// TIA Portal project "empty" (V15.1)

(* hardware
DEVICE "S7-1200 station_1"  S7-1200 Station
   slot 0: "Rack_0"  S7-1200 Rack  Rack  V1.0
   slot 1: "PLC_1"  CPU 1217C DC/DC/DC  6ES7 217-1AG40-0XB0  V4.1
*)

// ===== PLC "PLC_1"  CPU 1217C DC/DC/DC =====

VAR_GLOBAL   // PLC tag table "Default tag table"
   "b1_Pulse" AT %Q0.1 : Bool;
   "b1_Direction" AT %Q0.5 : Bool;
   "Tag_1" AT %M0.0 : Bool;
   "Tag_2" AT %M0.1 : Bool;
   "System_Byte" AT %MB0 : Byte;
   "FirstScan" AT %M0.0 : Bool;
   "DiagStatusUpdate" AT %M0.1 : Bool;
   "AlwaysTRUE" AT %M0.2 : Bool;
   "AlwaysFALSE" AT %M0.3 : Bool;
   "Clock_Byte" AT %MB1 : Byte;
   "Clock_10Hz" AT %M1.0 : Bool;
   "Clock_5Hz" AT %M1.1 : Bool;
   "Clock_2.5Hz" AT %M1.2 : Bool;
   "Clock_2Hz" AT %M1.3 : Bool;
   "Clock_1.25Hz" AT %M1.4 : Bool;
   "Clock_1Hz" AT %M1.5 : Bool;
   "Clock_0.625Hz" AT %M1.6 : Bool;
   "Clock_0.5Hz" AT %M1.7 : Bool;
END_VAR

DATA_BLOCK "b1"   // DB1, Motion_DB
{ S7_Optimized_Access := 'TRUE' }
AUTHOR : SIMATIC
FAMILY : BasicMC
NAME : TO_PosAx
VERSION : 5.0
// stored: InstanceOfName TO_PositioningAxis
"TO_PositioningAxis"
BEGIN
   // Axis.LengthUnitNormalized.Distance = 1005
   // Axis.DirectionOutputEnabledCU = TRUE
   // Axis.OnlinePtoModeCU = 16#0000_0002
   // Axis.SelectedChannel2EnumCU = %Q0.5
   // Axis.SelectedChannel1EnumCU = %Q0.1
   // Pulse.MinDeltaDeltaFrequencyCU = 0.004
   // Pulse.MaxDeltaDeltaFrequencyCU = 1.0E+10
   // Pulse.MinDeltaFrequencyCU = 0.005
   // Pulse.MaxDeltaFrequencyCU = 9.5E+9
   // Pulse.MinFrequencyCU = 1.0
   // Pulse.MaxFrequencyCU = 1.0E+6
   // Pulse.OutputSourceCU = 16#0000_0000
   // Axis.SelectPTO = 0
   // Axis.LengthUnit.LastDistance = 1005
END_DATA_BLOCK

ORGANIZATION_BLOCK "Main"   // OB1, LAD, ProgramCycle
TITLE = "Main Program Sweep (Cycle)"
{ S7_Optimized_Access := 'TRUE' }
VERSION : 0.1
   VAR_INPUT
      Initial_Call : Bool;   // Initial call of this OB
      Remanence : Bool;   // =True, if remanent data are available
   END_VAR
BEGIN

REGION Network 1
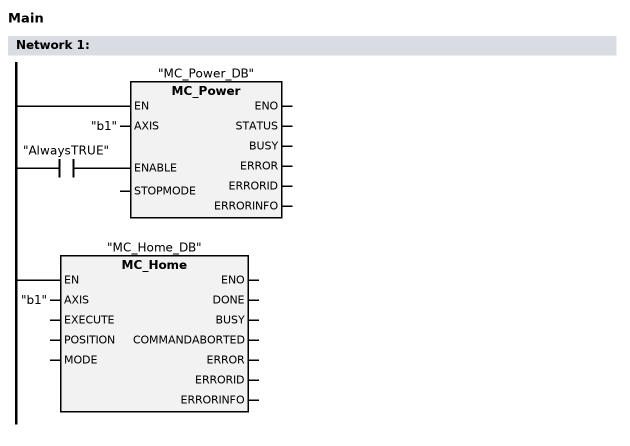
   "MC_Power_DB"(Axis := "b1", Enable := "AlwaysTRUE");   // MC_Power
   "MC_Home_DB"(Axis := "b1");   // MC_Home
END_REGION
END_ORGANIZATION_BLOCK